{attribute 'linkalways'} 
{attribute 'no_explicit_call' := 'This FB is a CLASS and must be accessed using methods or properties'}
{attribute 'enable_dynamic_creation'}
FUNCTION_BLOCK _Array0to7OfLREAL EXTENDS ArrayDatatypeBase_1D
VAR CONSTANT
	lBound : DINT := 0;
	uBound : DINT := 7;
END_VAR
VAR
	localData : ARRAY [lBound..uBound] OF LREAL;
	activeData : REFERENCE TO ARRAY [lBound..uBound] OF LREAL REF= localData;
	elements : ARRAY [lBound..uBound] OF _LREAL(0.0);
	baseType : _LREAL(0.0);
END_VAR

PROPERTY PUBLIC Address : PVOID
GET
Address := ADR(activeData);
END_GET
END_PROPERTY

PROPERTY PUBLIC BaseDatatype : I_Datatype
GET
BaseDatatype := baseType;
END_GET
END_PROPERTY

METHOD PUBLIC ClearReference
VAR_INPUT
END_VAR
activeData REF= localData;
SetElementReference();
END_METHOD

METHOD PUBLIC Clone : I_Datatype
VAR
    pClone : POINTER TO _Array0to7OfLREAL;
END_VAR
pClone := __NEW(_Array0to7OfLREAL());
pClone^.Value := Value;
Clone := pClone^;
END_METHOD

METHOD FB_init : BOOL
VAR_INPUT
	bInitRetains : BOOL; // if TRUE, the retain variables are initialized (warm start / cold start)
	bInCopyCode : BOOL;  // if TRUE, the instance afterwards gets moved into the copy code (online change)
END_VAR
SetElementReference();
END_METHOD

METHOD PUBLIC MakeReferenceTo
VAR_INPUT
	ReferenceTarget : REFERENCE TO ARRAY [lBound..uBound] OF LREAL;
END_VAR
activeData REF= ReferenceTarget;
SetElementReference();
END_METHOD

METHOD PROTECTED OnSerializeArrayValues
VAR_INPUT
	Serializer : I_Serializer;
END_VAR
VAR
	i : DINT;
END_VAR
FOR i := lBound TO uBound DO
	elements[i].SerializeWith(Serializer);
END_FOR
END_METHOD

METHOD PROTECTED SetElementReference
VAR_INPUT
END_VAR
VAR
	i : DINT;
END_VAR
FOR i := lBound TO uBound DO
	elements[i].MakeReferenceTo(activeData[i]);
END_FOR
END_METHOD

PROPERTY PUBLIC Size : UDINT
GET
Size := SIZEOF(activeData);
END_GET
END_PROPERTY

METHOD PROTECTED TryDeserializeArrayValues : BOOL
VAR_INPUT
	Deserializer : I_Deserializer;
	Feedback : I_DeserializerFeedback;
END_VAR
VAR
	enumerator : I_DeserializerArrayForwardEnumerator;
	i : DINT;
END_VAR
enumerator := Deserializer.GetArrayEnumerator();
i := lBound;

WHILE enumerator.MoveNext() AND i <= uBound DO
	
	IF NOT elements[i].TryDeserializeFrom(enumerator.Current, Feedback) THEN
		EXIT;
	END_IF
	i := i + 1;

END_WHILE
enumerator.Dispose();
END_METHOD

METHOD PUBLIC TryGetElementAsDatatypeByIndex : BOOL
VAR_INPUT
	Index : DINT;
	Destination : REFERENCE TO I_Datatype;
END_VAR
IF Index < lbound OR Index > ubound THEN
	RETURN;
END_IF

Destination := elements[Index];
TryGetElementAsDatatypeByIndex := TRUE;
END_METHOD

METHOD PUBLIC TryGetLowerBound : BOOL
VAR_INPUT
	Dimention : UDINT;
	Destination : REFERENCE TO DINT;
END_VAR
IF Dimention = 1 THEN
	Destination := lBound;
	TryGetLowerBound := TRUE;
END_IF
END_METHOD

METHOD PUBLIC TryGetUpperBound : BOOL
VAR_INPUT
	Dimention : UDINT;
	Destination : REFERENCE TO DINT;
END_VAR
IF Dimention = 1 THEN
	Destination := uBound;
	TryGetUpperBound := TRUE;
END_IF
END_METHOD

METHOD TryMakeReferenceTo : BOOL
VAR_INPUT
	Target : I_Datatype;
END_VAR
VAR
	targetAsArray : I_ArrayDatatype;
	pTargetData : POINTER TO ARRAY [lBound..uBound] OF LREAL;
END_VAR
IF NOT Target.TryResolveAsArrayDatatype(targetAsArray) THEN
	RETURN;
END_IF

IF NOT (targetAsArray.Identifier = Identifier) THEN
	RETURN;
END_IF

pTargetData := Target.Address;
activeData REF= pTargetData^;
SetElementReference();
TryMakeReferenceTo := TRUE;
END_METHOD

PROPERTY PUBLIC Value : REFERENCE TO ARRAY [lBound..uBound] OF LREAL;
GET
Value ref= activeData;
END_GET
END_PROPERTY

END_FUNCTION_BLOCK

(* stored: Version 1.1.0.1, ProductVersion 3.1.4024.13
   POU _Array0to7OfLREAL: Id {1679230a-e763-064c-273c-fae0ea399d95}, SpecialFunc None
   Folder Core: Id {fd1f63d7-2898-0703-0b52-94efc3e7645d}
   Folder Constructor: Id {5845d816-245e-03bd-39e9-3ed1b0d8d39a}
   Folder Protected: Id {064900f7-8f79-0886-2d3a-8cf95bfa83a4}
   Folder Customize: Id {04f7a8c7-0daa-095b-060a-c80f46a1a7ad}
   Property Address: Id {431328dd-8ef5-0f3a-1bc8-504c20d38bfc}
   Get Get: Id {f0e2c166-a939-080a-2c13-5347bab6ca85}
   Property BaseDatatype: Id {74500aab-5cdb-01fb-1ff2-1409d6b13e05}
   Get Get: Id {97ec7d4a-9f90-09e1-3fa8-23060e897bff}
   Method ClearReference: Id {17c0f5f4-3318-06a2-1b12-c9ad72fe9fee}
   Method Clone: Id {c54a1d61-f955-0545-1b55-09b7c5898e3f}
   Method FB_init: Id {e9c1a768-13ad-0f61-3fac-3f5395708cdb}
   Method MakeReferenceTo: Id {96f6d617-c4e4-09ec-380f-7eccac0a371c}
   Method OnSerializeArrayValues: Id {6b840c9e-2195-0a2e-27ef-6f3fd8543b39}
   Method SetElementReference: Id {a6362c6d-b4cc-0b15-012b-66229abfb774}
   Property Size: Id {cedbf395-44ae-003a-2d68-ff1f1681b3e1}
   Get Get: Id {b2b46b07-2fe4-0042-33c2-99cb8bfa8043}
   Method TryDeserializeArrayValues: Id {ef9cefac-eedc-04ce-1db4-05273dfc61ac}
   Method TryGetElementAsDatatypeByIndex: Id {62e896cf-af36-0083-114b-f5e5cfd1e2b3}
   Method TryGetLowerBound: Id {2bedff98-a3fd-0784-0e0b-6a899db81e6d}
   Method TryGetUpperBound: Id {17420a90-d841-094f-385d-36db9e5feb84}
   Method TryMakeReferenceTo: Id {e4d9da29-e45d-0f6e-1c34-9db3f1ba0553}
   Property Value: Id {40a41487-8e0c-0a61-2af9-9aefaca12431}
   Get Get: Id {cef17429-e599-01f8-3582-6b79b51572ee} *)
